(* PLC project DM1ErrorTexts, Hydac System GmbH PdtCodeBuilder.dll 1.2.7.80 *)
(* stored: companyURL http://www.hydac.com/, contentDescription This content was automatically generated. Please do not edit., creationDateTime 2025-04-18T16:40:50.760 *)

VAR_GLOBAL CONSTANT  (* DM1ErrorTexts *)
  DM1_LANGUAGE_COUNT : INT := 3;
  g_DM1Texts_NativeLanguageName : ARRAY[0..2] OF WSTRING(7) := ["german", "english", "french"];
  DM1_FMI_COUNT : INT := 33;
  g_DM1Texts_FMI : ARRAY[0..2, 0..32] OF WSTRING(40) := ["Signal extrem hoch, kritisch", "Signal extrem niedrig, kritisch", "Daten fehlerhaft o. nicht plausibel", "Kurzschluß zu Plus / Spannung hoch", "Kurzschluß zu Masse / Spannung gering", "Kabelbruch / Strom gering", "Kurzschluß nach Masse / Strom hoch", "Mechanik reag. nicht / klemmt betätigt", "Anormale Frequenz, Pulsweite o. Periode", "Zeitüberschreitung / anormale Taktrate", "Anormale Änderungsgeschwindigkeit", "Fehlerursache nicht bekannt", "Steuergerät interner Fehler ", "Ausserhalb der Kalibirierung", "Spezielle Anleitung", "Signal zu hoch", "Signal sehr hoch", "Signal zu niedrig", "Signal sehr niedrig", "Datenempfang mit aktiven Fehlerstatus", "Werte driften hoch", "Werte driften runter", "Kein Signal / Bauteil fehlt", "Nicht Kalibriert", "Logischer Fehler (SW Fehler)", "Klemmt offen", "Ausserhalb gültigen Wertebreichs", "Kabelbruch o. Kurzschluß n. Masse", "Kabelbruch o. Kurzschluß n. Plus", "Reserve", "Reserve", "Fehlerzustand laut SPN", "FMI_NONE", "Signal Very High Critical", "Signal Very Low Critical", "Data erratic or intermittent", "Short to Power (Voltage High)", "Short to Ground (Voltage Low)", "Open Circuit (Current Low)", "Short to Ground (Current High)", "Mechanic not responding / Stuck Actuated", "Abnormal Freque., Pulse Width or Period", "Timeout / Abnormale update rate", "Abnormal rate of change", "Error root cause not known", "Internal Controller Error", "Out of Calibration", "Special Instructions", "Signal too High", "Signal very High", "Signal too Low", "Signal very Low", "Received Data with Active Error State", "Data drifted high", "Data drifted low", "No Signal / Component Missing", "Not Calibrated", "Logical Error (SW Failure)", "Stuck Open", "Out of Valid Range", "Open Circuit or Short to Ground", "Open Circuit or Short to Power", "Reserve", "Reserve", "Error condition exists according to SPN ", "FMI_NONE", "Signal tres haut critique", "Signal tres bas critique", "Erreur de donées", "Haute tension / Court-circuit a batterie", "Basse tension / Court-circuit a masse", "Courant bas / non connecté", "Courant haut / Court-circuit a masse", "Mécanique ne response pas/ Bloquer fermé", "Anormal fréqu., duree d'impuls., période", "Depasment Temps / Anormal débit transm.", "Anormal vitesse de changement", "Origine de l'erreur inconnu", "Erreur interne a l'ECU", "Hors calibration", "Instruction spécial", "Signal trop haut", "Signal tres haut", "Signal trop bas", "Signal tres bas", "Reception d'erreurs sur les données", "Valeurs dériver en haut", "Valeurs dériver en bas", "Pas de signal / Élément absent ", "Pas calibré", "Erreur de logique / Logiciel", "Bloquer ouvert", "Hors valide domain des valeurs", "Non connecté ou Court-circuit a masse", "Non connecté ou Court-circuit a batterie", "Reserve", "Reserve", "Condition erreur correspondante a SPN", "FMI_NONE"];
  DM1_FMIEX_COUNT : INT := 1;
  g_DM1Texts_FMIEX : ARRAY[0..2, 0..0] OF WSTRING(10) := ["FMIEX_NONE", "FMIEX_NONE", "FMIEX_NONE"];
  DM1_ASSEMBLY_COUNT : INT := 1;
  g_DM1Texts_Assembly : ARRAY[0..2, 0..0] OF WSTRING(8) := ["ASM_NONE", "ASM_NONE", "ASM_NONE"];
  DM1_COMPONENTTYPE_COUNT : INT := 1;
  g_DM1Texts_ComponentType : ARRAY[0..2, 0..0] OF WSTRING(9) := ["COMP_NONE", "COMP_NONE", "COMP_NONE"];
  DM1_COMPONENTFUNCTION_COUNT : INT := 18;
  g_DM1Texts_ComponentFunction : ARRAY[0..2, 0..17] OF WSTRING(31) := ["NV_PARAMERTERS_C0", "NV_PARAM_SPEED_MAX_RAIL", "NV_PARAM_BRAKE_TEST", "NV_PARAM_RAIL_WORK_SAFETY_C0", "NV_PARAM_TRANSPORT_POS_C0", "NV_PARAM_SELECT_CONTROL_POST", "NV_PARAM_ALARM_C0", "NV_PARAM_MAST_DISPLAY", "NV_PARAMERTERS_C1", "NV_PARAM_MOTOR_C1", "NV_PARAM_LIMIT_WORK_ENVELOPE_C1", "NV_PARAM_MVT_END_STOP_C1", "NV_PARAM_AUTO_STOP_C1", "NV_PARAM_MAST_C1", "NV_PARAM_ALARM_C1", "NV_OPTION_C0", "NV_OPTION_C1", "FUNC_NONE", "NV_PARAMERTERS_C0", "NV_PARAM_SPEED_MAX_RAIL", "NV_PARAM_BRAKE_TEST", "NV_PARAM_RAIL_WORK_SAFETY_C0", "NV_PARAM_TRANSPORT_POS_C0", "NV_PARAM_SELECT_CONTROL_POST", "NV_PARAM_ALARM_C0", "NV_PARAM_MAST_DISPLAY", "NV_PARAMERTERS_C1", "NV_PARAM_MOTOR_C1", "NV_PARAM_LIMIT_WORK_ENVELOPE_C1", "NV_PARAM_MVT_END_STOP_C1", "NV_PARAM_AUTO_STOP_C1", "NV_PARAM_MAST_C1", "NV_PARAM_ALARM_C1", "NV_OPTION_C0", "NV_OPTION_C1", "FUNC_NONE", "NV_PARAMERTERS_C0", "NV_PARAM_SPEED_MAX_RAIL", "NV_PARAM_BRAKE_TEST", "NV_PARAM_RAIL_WORK_SAFETY_C0", "NV_PARAM_TRANSPORT_POS_C0", "NV_PARAM_SELECT_CONTROL_POST", "NV_PARAM_ALARM_C0", "NV_PARAM_MAST_DISPLAY", "NV_PARAMERTERS_C1", "NV_PARAMERTERS_C1", "NV_PARAM_MOTOR_C1", "NV_PARAM_LIMIT_WORK_ENVELOPE_C1", "NV_PARAM_MVT_END_STOP_C1", "NV_PARAM_AUTO_STOP_C1", "NV_PARAM_ALARM_C1", "NV_OPTION_C0", "NV_OPTION_C1", "FUNC_NONE"];
  DM1_SPN_SRC_COUNT_New_Master_List : INT := 1194;
